(* Logix 5000 project; controller SOCK vendor 1 type 14 code 92 rev 20.56; software revision 20.00 *)

TASK MainTask (periodic, rate 20 ms, priority 10, watchdog 500 ms) : Process

MODULES
   Local : vendor 1 type 14 code 92 (ICP 0, rev 20.56)
      A1_AD2 : vendor 1 type 12 code 200 (ICP 1, Ethernet 172.16.3.121, rev 10.7, Input RPI 500 ms)
      A1_AD3 : vendor 1 type 12 code 200 (Ethernet 172.16.3.123, ICP 2, rev 10.7, Input RPI 500 ms)
END_MODULES

TYPE AcceptResponse :
STRUCT
   Instance : DINT;
   Addr : SockAddr;
END_STRUCT
END_TYPE

TYPE Anpars :
STRUCT
   Tg_inN1 : TAnpar;
   Tg_inAVO1 : TAnpar;
   Tg_outAVO1 : TAnpar;
   Tg_outN1 : TAnpar;
   Tg_inN2 : TAnpar;
   Tg_inAVO2 : TAnpar;
   Tg_outAVO2 : TAnpar;
   Tg_outN2 : TAnpar;
   Pg_aftKr4 : TAnpar;
   Pg_outSep21 : TAnpar;
   Pg_aftKr6 : TAnpar;
   Pg_aftKr16 : TAnpar;
   Pg_outSep22 : TAnpar;
   Pg_aftKr18 : TAnpar;
   dPg_Kr1 : TAnpar;
   dPg_Sep11 : TAnpar;
   dPg_Kr3 : TAnpar;
   dPg_AVO1 : TAnpar;
   dPg_Sep21 : TAnpar;
   dPg_Kr13 : TAnpar;
END_STRUCT
END_TYPE

TYPE OpenConnParam :
STRUCT
   Timeout : DINT;
   DestAddr : STRING;
END_STRUCT
END_TYPE

TYPE READ_DATA_REQ :
STRUCT
   Timeout : DINT;
   BufLen : DINT;
END_STRUCT
END_TYPE

TYPE READ_RESP :
STRUCT
   FromAddr : SockAddr;
   READ_BUFF : STR_4096;
END_STRUCT
END_TYPE

TYPE REQUEST_PARAMETERS :
STRUCT
   Type : DINT;   // 1 - TCP 2- UPD
   Addr : SockAddr;
END_STRUCT
END_TYPE

TYPE SockAddr :
STRUCT
   Family : INT;   // Address Family Must be 2
   Port : INT;   // Port Number
   Addr : DINT;   // IP Address
END_STRUCT
END_TYPE

TYPE SocketData :
STRUCT
   Instance : DINT;
   Attr : SocketInstAttr;
END_STRUCT
END_TYPE

TYPE SocketInstAttr :
STRUCT
   LocalAddr : SockAddr;
   RemoteAddr : SockAddr;
   SendBufSize : DINT;
   RcvBufSize : DINT;
   TCPKeepAlive : DINT;
   TCPNoDelay : DINT;
   InactivityTimeout : DINT;
   MulticastTTL : DINT;
   UDPBroadcast : DINT;
   LingerOnOff : DINT;
END_STRUCT
END_TYPE

TYPE STR_4096 :
STRUCT
   LEN : DINT;
   DATA : SINT[4096];
END_STRUCT
END_TYPE

TYPE STR_480 :
STRUCT
   LEN : DINT;
   DATA : SINT[480];
END_STRUCT
END_TYPE

TYPE TAnpar :
STRUCT
   Sys : REAL;
   Params : INT;
END_STRUCT
END_TYPE

TYPE TFastRetroBuf :
STRUCT
   LEN : DINT;
   PacketSize : DINT;
   Data : REAL[109];
END_STRUCT
END_TYPE

TYPE Write_Data :
STRUCT
   Timeout : DINT;
   ToAddr : SockAddr;
   BufLen : DINT;
   Buf : SINT[20];
END_STRUCT
END_TYPE

TYPE WRT_DATA :
STRUCT
   Timeout : DINT;
   ToAddr : SockAddr;
   Buffer : TFastRetroBuf;
END_STRUCT
END_TYPE

ADD_ON_INSTRUCTION _FastRetro_checkErr   (* revision 1.0 *)
// Проверка ошибок в сообщении, возвращает true, если необходимо предпринять действия
VAR_IN_OUT
   Msg : MESSAGE; {required}
END_VAR
VAR_OUTPUT
   err : DINT; {required}   // Принятие решений 0-не треб., 1-отвалился сокет, 10-другое
END_VAR
VAR_IN_OUT
   errCount : DINT; {required}
END_VAR

ROUTINE Logic   (* structured text *)
   err := 0;
   if(Msg.ER) then
   	if(errCount > 3) then
   		//что-то делаем при ошибке отправки
   		//16#0000_0036 - Соединение принудительно закрыто клиентом, рекоммендация - удалить сокет и поробовать восстановить
   		if(Msg.EXERR = 16#0000_0036
   			or Msg.EXERR = 16#0000_0033 ) then //Обрыв связи
   			err := 1;
   		else
   			err := 10;
   		end_if;
   		//обнуляем хендл соответствующего сокета, так как теперь мы его удаляем (state = 13)
   	end_if;
   else
   	errCount := 0;
   end_if;
END_ROUTINE
END_ADD_ON_INSTRUCTION

ADD_ON_INSTRUCTION _test   (* revision 1.0 *)
// Проверка ошибок в сообщении, возвращает true, если необходимо предпринять действия
VAR_IN_OUT
   Msg : MESSAGE; {required}
END_VAR
VAR_OUTPUT
   err : DINT; {required}   // Принятие решений 0-не треб., 1-отвалился сокет, 10-другое
END_VAR
VAR_IN_OUT
   errCount : DINT; {required}
END_VAR

ROUTINE Logic   (* structured text *)
   err := 0;
   if(Msg.ER) then
   	if(errCount > 3) then
   		//что-то делаем при ошибке отправки
   		//16#0000_0036 - Соединение принудительно закрыто клиентом, рекоммендация - удалить сокет и поробовать восстановить
   		if(Msg.EXERR = 16#0000_0036
   			or Msg.EXERR = 16#0000_0033 ) then //Обрыв связи
   			err := 1;
   		else
   			err := 10;
   		end_if;
   		//обнуляем хендл соответствующего сокета, так как теперь мы его удаляем (state = 13)
   	end_if;
   else
   	errCount := 0;
   end_if;
END_ROUTINE
END_ADD_ON_INSTRUCTION

VAR_GLOBAL   (* controller tags *)
   _EWEB_PATH : STRING := '$01$01';
   AcceptReqTimer : FBD_TIMER;
   Anpar : Anpars;
   BufLenSent : DINT := 7;
   Change_Log_Msg : MESSAGE;
        MessageParameters(ServiceCode := 16#0010, LocalElement := Log_enable, ...)
   CLOCK : DINT[7] := ([0] := 1998, [1] := 1, [2] := 12, [3] := 22, [4] := 11, [5] := 13, [6] := 576094);
   COLN : STRING := ':';
   Conn_Accept_MSG : MESSAGE;
        MessageParameters(ServiceCode := 16#0050, LocalElement := Sock_Accept_Timeout, DestinationTag := Sock_Accept_Resp, ...)
   Create_Sock_MSG : MESSAGE;
        MessageParameters(ServiceCode := 16#004b, LocalElement := Socket, DestinationTag := Instance, ...)
   Delete_All_MSG : MESSAGE;
        MessageParameters(ServiceCode := 16#0051, ...)
   Delete_Sock_MSG : MESSAGE;
        MessageParameters(ServiceCode := 16#004f, ...)
   Enable_Log_MSG : MESSAGE;
        MessageParameters(ServiceCode := 16#000e, DestinationTag := Log_enable, ...)
   Get_Sock_Object_MSG : MESSAGE;
        MessageParameters(ServiceCode := 16#0001, DestinationTag := Socket_Object_Class_Response[0], ...)
   Get_SockTimeout_MSG : MESSAGE;
        MessageParameters(ServiceCode := 16#000e, DestinationTag := SockTimeout, ...)
   HOUR : STRING := '22';
   Instance : DINT := 484;
   Log_enable : DINT;
   Log_old : DINT;
   MINUTE : STRING := '11';
   Read_Data_MSG : MESSAGE;
        MessageParameters(ServiceCode := 16#004d, LocalElement := Read_Data_Req, DestinationTag := Read_Response, ...)
   Read_Data_Req : READ_DATA_REQ := (Timeout := 1000, BufLen := 100);
   Read_Response : READ_RESP := (READ_BUFF := '07:50:1207:50:1307:50:14');
   SECOND : STRING := '13';
   Set_SockTimeout_MSG : MESSAGE;
        MessageParameters(ServiceCode := 16#0010, LocalElement := SockTimeout, ...)
   Sock_Accept_Resp : AcceptResponse := (Instance := 4805, Addr.Family := 2, Addr.Port := 1188, Addr.Addr := 1684298241);
   Sock_Accept_Timeout : DINT := 26000;
   Sock_Object_Data : DINT[13] := ([0] := 655425538, [4] := 2048, [5] := 2048, [6] := 8, [7] := 1, [8] := 300000);
   Socket : REQUEST_PARAMETERS := (Type := 1, Addr.Family := 2, Addr.Port := 10000);
   Socket_Object_Class_Response : SINT[10] := ([0] := 1, [2] := 20);
   SockTimeout : DINT;
   TIME : STRING := '22:11:13';
   Write_Data_MSG : MESSAGE;
        MessageParameters(ServiceCode := 16#004e, LocalElement := Write_Data_Out, DestinationTag := BufLenSent, ...)
   Write_Data_MSG_RED : MESSAGE;
        MessageParameters(ServiceCode := 16#004e, LocalElement := Write_Data_Out, DestinationTag := BufLenSent, ...)
   Write_Data_Out : WRT_DATA := (Timeout := 20000, ToAddr.Family := 2);
   zero : STRING := '0';
END_VAR

PROGRAM _Remove
VAR
   _FastRetro_checkErr : _test;
   Accept : ALIAS FOR Log_Enable.2;
   Accept_Request : BOOL;   // Toggle this Bit to Accept Incoming Connection
   Attrubute : ALIAS FOR Log_Enable.6;
   ClientsId : SocketData[10];
   ClientsIdSize : DINT;
   CommonErrors : DINT;
   ConnCount : DINT;
   Create : ALIAS FOR Log_Enable.0;
   Create_Socket_Req : BOOL;
   CreatedPacketsCount : DINT;
   CurStatusFlagsWrite : DINT;
   CycleNumber : DINT;
   Delete : ALIAS FOR Log_Enable.5;
   Delete_All_Request : BOOL;
   Delete_Sockets_Req : BOOL;
   ElementsCount : DINT;
   Enable_Log_Req : BOOL;
   Err_Write_Red : DINT;
   errCntWriteMain : DINT;
   errCntWriteRed : DINT;
   errCode : DINT;   // Код ошибки
   Errors : ALIAS FOR Log_Enable.7;
   FirstPacketSendMain : BOOL;
   FirstPacketSendRed : BOOL;
   frontSend : BOOL;
   Get_Socket_Instance_Req : BOOL;
   Get_Socket_Object_Req : BOOL;
   Get_SocketTimeout : BOOL;
   increment : DINT;
   isCurSockMain : BOOL;
   it : DINT;
   iter : DINT;
   Log_Enable : DINT := 255;
   loseCyclesCount : DINT;
   MainMsg : DINT; {constant, access Read Only}   // Константа = 0
   MaxCyclesCount : DINT;
   needToResend : BOOL;
   Nothing : BOOL := 1;
   Open : ALIAS FOR Log_Enable.1;
   ParCount : DINT;
   point : REAL;
   Read : ALIAS FOR Log_Enable.3;
   Read_Data_Request : BOOL;   // Toggle This Bit to Read Incoming Data
   RedMsg : DINT := 1; {constant, access Read Only}   // Константа = 1
   SendPacketsCount : DINT;
   serverState : DINT;
   Set_SocketTimeout : BOOL;
   SockInstance : DINT;
   systemDataCount : DINT;
   tcpserverInit : BOOL;
   TempBuffer : REAL[400];
   Write : ALIAS FOR Log_Enable.4;
   Write_Request : BOOL;
END_VAR
END_PROGRAM

PROGRAM MainProgram   (* main routine TCP_Server *)
VAR
   _FastRetro_checkErr : _FastRetro_checkErr;
   Accept : ALIAS FOR Log_Enable.2;
   Accept_Request : BOOL;   // Toggle this Bit to Accept Incoming Connection
   Attrubute : ALIAS FOR Log_Enable.6;
   ClientsId : SocketData[10];
   ClientsIdSize : DINT;
   CommonErrors : DINT;
   ConnCount : DINT;
   Create : ALIAS FOR Log_Enable.0;
   Create_Socket_Req : BOOL;
   CreatedPacketsCount : DINT;
   CurStatusFlagsWrite : DINT;
   CycleNumber : DINT;
   Delete : ALIAS FOR Log_Enable.5;
   Delete_All_Request : BOOL;
   Delete_Sockets_Req : BOOL;
   ElementsCount : DINT;
   Enable_Log_Req : BOOL;
   Err_Write_Red : DINT;
   errCntWriteMain : DINT;
   errCntWriteRed : DINT;
   errCode : DINT;   // Код ошибки
   Errors : ALIAS FOR Log_Enable.7;
   FirstPacketSendMain : BOOL;
   FirstPacketSendRed : BOOL;
   frontSend : BOOL;
   Get_Socket_Instance_Req : BOOL;
   Get_Socket_Object_Req : BOOL;
   Get_SocketTimeout : BOOL;
   increment : DINT;
   isCurSockMain : BOOL;
   it : DINT;
   iter : DINT;
   Log_Enable : DINT := 255;
   loseCyclesCount : DINT;
   MainMsg : DINT; {constant, access Read Only}   // Константа = 0
   MaxCyclesCount : DINT;
   needToResend : BOOL;
   Nothing : BOOL := 1;
   Open : ALIAS FOR Log_Enable.1;
   ParCount : DINT;
   point : REAL;
   Read : ALIAS FOR Log_Enable.3;
   Read_Data_Request : BOOL;   // Toggle This Bit to Read Incoming Data
   RedMsg : DINT := 1; {constant, access Read Only}   // Константа = 1
   SendPacketsCount : DINT;
   serverState : DINT;
   Set_SocketTimeout : BOOL;
   SockInstance : DINT;
   systemDataCount : DINT;
   tcpserverInit : BOOL;
   TempBuffer : REAL[400];
   Write : ALIAS FOR Log_Enable.4;
   Write_Request : BOOL;
END_VAR

ROUTINE _SOCKET_ATTR   (* ladder *)
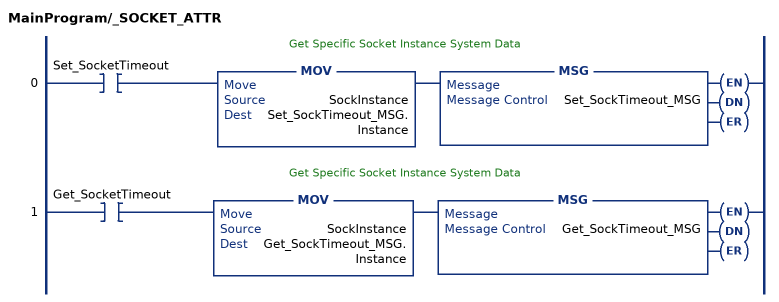
   // Get Specific Socket Instance System Data
   0: XIC(Set_SocketTimeout)MOV(SockInstance,Set_SockTimeout_MSG.Instance)MSG(Set_SockTimeout_MSG);
   // Get Specific Socket Instance System Data
   1: XIC(Get_SocketTimeout)MOV(SockInstance,Get_SockTimeout_MSG.Instance)MSG(Get_SockTimeout_MSG);
END_ROUTINE

ROUTINE _SOCKET_STATS   (* ladder *)
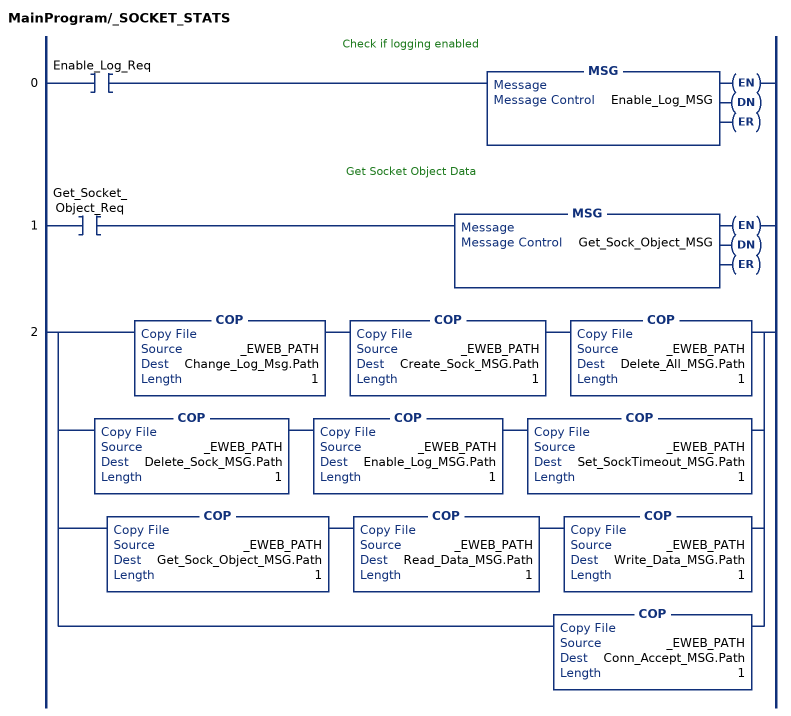
   // Check if logging enabled
   0: XIC(Enable_Log_Req)MSG(Enable_Log_MSG);
   // Get Socket Object Data
   1: XIC(Get_Socket_Object_Req)MSG(Get_Sock_Object_MSG);
   2: [COP(_EWEB_PATH,Change_Log_Msg.Path,1) COP(_EWEB_PATH,Create_Sock_MSG.Path,1) COP(_EWEB_PATH,Delete_All_MSG.Path,1) ,COP(_EWEB_PATH,Delete_Sock_MSG.Path,1) COP(_EWEB_PATH,Enable_Log_MSG.Path,1) COP(_EWEB_PATH,Set_SockTimeout_MSG.Path,1) ,COP(_EWEB_PATH,Get_Sock_Object_MSG.Path,1) COP(_EWEB_PATH,Read_Data_MSG.Path,1) COP(_EWEB_PATH,Write_Data_MSG.Path,1) ,COP(_EWEB_PATH,Conn_Accept_MSG.Path,1) ];
END_ROUTINE

ROUTINE _SOCKET_TCP_SERV   (* ladder *)
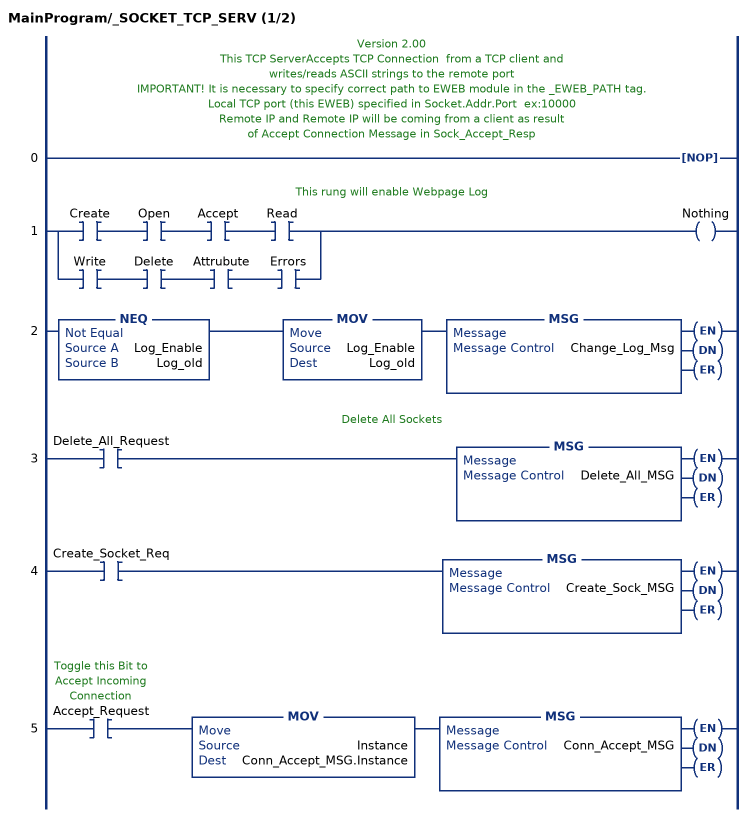
   // Version 2.00
   // This TCP ServerAccepts TCP Connection  from a TCP client and
   // writes/reads ASCII strings to the remote port
   // IMPORTANT! It is necessary to specify correct path to EWEB module in the _EWEB_PATH tag.
   // Local TCP port (this EWEB) specified in Socket.Addr.Port  ex:10000
   // Remote IP and Remote IP will be coming from a client as result
   // of Accept Connection Message in Sock_Accept_Resp
   0: NOP();
   // This rung will enable Webpage Log
   1: [XIC(Create) XIC(Open) XIC(Accept) XIC(Read) ,XIC(Write) XIC(Delete) XIC(Attrubute) XIC(Errors) ]OTE(Nothing);
   2: NEQ(Log_Enable,Log_old)MOV(Log_Enable,Log_old)MSG(Change_Log_Msg);
   // Delete All Sockets
   3: XIC(Delete_All_Request)MSG(Delete_All_MSG);
   4: XIC(Create_Socket_Req)MSG(Create_Sock_MSG);
   5: XIC(Accept_Request)MOV(Instance,Conn_Accept_MSG.Instance)MSG(Conn_Accept_MSG);
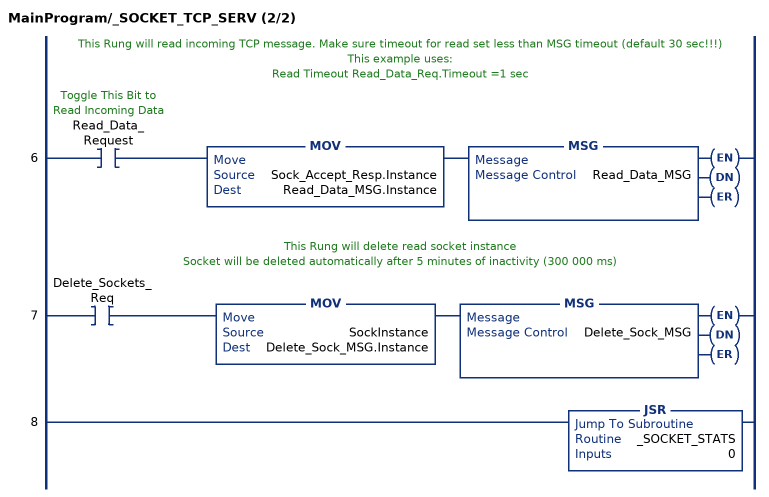
   // This Rung will read incoming TCP message. Make sure timeout for read set less than MSG timeout (default 30 sec!!!)
   // This example uses:
   // Read Timeout Read_Data_Req.Timeout =1 sec
   6: XIC(Read_Data_Request)MOV(Sock_Accept_Resp.Instance,Read_Data_MSG.Instance)MSG(Read_Data_MSG);
   // This Rung will delete read socket instance
   // Socket will be deleted automatically after 5 minutes of inactivity (300 000 ms)
   7: XIC(Delete_Sockets_Req)MOV(SockInstance,Delete_Sock_MSG.Instance)MSG(Delete_Sock_MSG);
   8: JSR(_SOCKET_STATS,0);
END_ROUTINE

ROUTINE _SOCKET_WRITE_MAIN   (* ladder *)
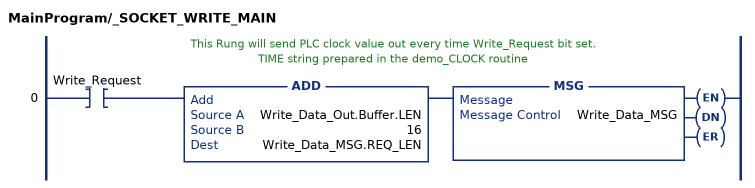
   // This Rung will send PLC clock value out every time Write_Request bit set.
   // TIME string prepared in the demo_CLOCK routine
   0: XIC(Write_Request)ADD(Write_Data_Out.Buffer.LEN,16,Write_Data_MSG.REQ_LEN)MSG(Write_Data_MSG);
END_ROUTINE

ROUTINE _SOCKET_WRITE_RED   (* ladder *)
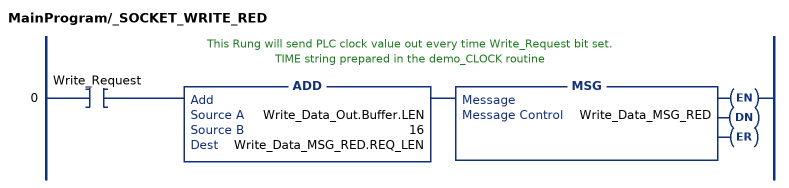
   // This Rung will send PLC clock value out every time Write_Request bit set.
   // TIME string prepared in the demo_CLOCK routine
   0: XIC(Write_Request)ADD(Write_Data_Out.Buffer.LEN,16,Write_Data_MSG_RED.REQ_LEN)MSG(Write_Data_MSG_RED);
END_ROUTINE

ROUTINE Exchange   (* structured text *)
   //Обрабатывается, когда сервер находится в состояниях 2-3
   
   /*
   	Заполнение данных в буфер передачи
   */
   GSV(WALLCLOCKTIME,,DateTime,CLOCK[0]);
   
   //на первом цикле заполняем служебный заголовок пакета
   if(CycleNumber=0) then
   	//дата - год месяц число
   	TempBuffer[0]:= CLOCK[0];
   	TempBuffer[1]:= CLOCK[1];
   	TempBuffer[2]:= CLOCK[2];
   	//время - часы минуты секунды микросекунды
   	TempBuffer[3]:= CLOCK[3];
   	TempBuffer[4]:= CLOCK[4];
   	TempBuffer[5]:= CLOCK[5];
   	TempBuffer[6]:= CLOCK[6];
   	//кол-во параметров
   	TempBuffer[7]:= ParCount;
   	//кол-во циклов для сбора данных
   	TempBuffer[8]:= MaxCyclesCount;
   	(*
   	//дата - год месяц число
   	Write_Data_Out.Buffer.Data[0]:= CLOCK[0];
   	Write_Data_Out.Buffer.Data[1]:= CLOCK[1];
   	Write_Data_Out.Buffer.Data[2]:= CLOCK[2];
   	//время - часы минуты секунды микросекунды
   	Write_Data_Out.Buffer.Data[3]:= CLOCK[3];
   	Write_Data_Out.Buffer.Data[4]:= CLOCK[4];
   	Write_Data_Out.Buffer.Data[5]:= CLOCK[5];
   	Write_Data_Out.Buffer.Data[6]:= CLOCK[6];
   	Write_Data_Out.Buffer.Data[7]:= ParCount;
   	Write_Data_Out.Buffer.Data[8]:= MaxCyclesCount;
   	*)
   end_if;
   
   /*
   ! 	Заполняется пользователем ( правая часть, после := )
   	Порядок следования параметров должен совпадать с описанными в signals.ini (идет в комплекте с FastRetroApp)
   */
   if(CycleNumber<5 and ParCount<=20) then
   	TempBuffer[ParCount*CycleNumber+1+systemDataCount] := Anpar.Tg_inN1.Sys;
   	TempBuffer[ParCount*CycleNumber+2+systemDataCount] := Anpar.Tg_inAVO1.Sys;
   	TempBuffer[ParCount*CycleNumber+3+systemDataCount] := Anpar.Tg_outAVO1.Sys;
   	TempBuffer[ParCount*CycleNumber+4+systemDataCount] := Anpar.Tg_outN1.Sys;
   	TempBuffer[ParCount*CycleNumber+5+systemDataCount] := Anpar.Tg_inN2.Sys;
   	TempBuffer[ParCount*CycleNumber+6+systemDataCount] := Anpar.Tg_inAVO2.Sys;
   	TempBuffer[ParCount*CycleNumber+7+systemDataCount] := Anpar.Tg_outAVO2.Sys;
   	TempBuffer[ParCount*CycleNumber+8+systemDataCount] := Anpar.Tg_outN2.Sys;
   	TempBuffer[ParCount*CycleNumber+9+systemDataCount] := Anpar.Pg_aftKr4.Sys;
   	TempBuffer[ParCount*CycleNumber+10+systemDataCount] := Anpar.Pg_outSep21.Sys;
   	TempBuffer[ParCount*CycleNumber+11+systemDataCount] := Anpar.Pg_aftKr6.Sys;
   	TempBuffer[ParCount*CycleNumber+12+systemDataCount] := Anpar.Pg_aftKr16.Sys;
   	/*
   	TempBuffer[ParCount*CycleNumber+13+systemDataCount] := Anpar.Pg_outSep22.Sys;
   	TempBuffer[ParCount*CycleNumber+14+systemDataCount] := Anpar.Pg_aftKr18.Sys;
   	TempBuffer[ParCount*CycleNumber+15+systemDataCount] := Anpar.dPg_Kr1.Sys;
   	TempBuffer[ParCount*CycleNumber+16+systemDataCount] := Anpar.dPg_Sep11.Sys;
   	TempBuffer[ParCount*CycleNumber+17+systemDataCount] := Anpar.dPg_Kr3.Sys;
   	TempBuffer[ParCount*CycleNumber+18+systemDataCount] := Anpar.dPg_AVO1.Sys;
   	TempBuffer[ParCount*CycleNumber+19+systemDataCount] := Anpar.dPg_Sep21.Sys;
   	TempBuffer[ParCount*CycleNumber+20+systemDataCount] := Anpar.dPg_Kr13.Sys;
   	*/
   else
   	//исп. для отладки
   	loseCyclesCount := loseCyclesCount + 1;
   end_if;
   
   //чтобы предотвратить бесконечный рост CycleNumber
   if(CycleNumber < (MaxCyclesCount + 5)) then
   	CycleNumber := CycleNumber + 1;
   end_if;
   
END_ROUTINE

ROUTINE SendMessage   (* structured text *)
   COP(TempBuffer[0],Write_Data_Out.Buffer.Data[0],ElementsCount);
   //количество сформированных пакетов
   //CreatedPacketsCount := CreatedPacketsCount + 1;
   if(Write_Data_MSG.ER and (ClientsId[MainMsg].Instance>0)) then
   	errCntWriteMain := errCntWriteMain + 1;
   elsif(Write_Data_MSG_RED.ER and (ClientsId[RedMsg].Instance>0)) then
   	errCntWriteRed := errCntWriteRed + 1;
   end_if;
   if(ClientsId[MainMsg].Instance>0) then
   	FirstPacketSendMain := 1;
   end_if;
   if(ClientsId[RedMsg].Instance>0) then
   	FirstPacketSendRed := 1;
   end_if;
   
   Write_Request := 1;
   CycleNumber := 0;
   //NeedToSend.TimerEnable := 0;
   needToResend := 0;
END_ROUTINE

ROUTINE SocketInit   (* structured text *)
   if(isCurSockMain) then
   	SockInstance := ClientsId[MainMsg].Instance;
   else
   	SockInstance := ClientsId[RedMsg].Instance;
   end_if;
   
   //по умолчанию ставим 30 секунд таймаут безактивности
   SockTimeout := 30000;
   Set_SocketTimeout := 1;
   
   JSR(_SOCKET_ATTR);
   
   Set_SocketTimeout := 0;
   
   Get_SocketTimeout := 1;
   JSR(_SOCKET_ATTR);
   Get_SocketTimeout := 0;
END_ROUTINE

ROUTINE TCP_Server   (* structured text *)
   // 	версия 1.0
   /*
   	отправка сообщений асинхронная, поэтому флаги актуально
   	копировать в переменную в начале цикла:
   	.2 - .EW
   	.4 - .ER
   	.5 - .DN
   	.6 - .ST
   	.7 - .EN
   	.8 - .TO
   	.9 - .EN_CC
   */
   CurStatusFlagsWrite := Write_Data_MSG.Flags;
   
   //инициализационные параметры.
   if (not tcpserverInit) then
   
   //! заполняются пользователем
   
   	//количество параметров
   	ParCount := 12;
   //!
   	/*
   		Кол-во циклов в посылке для текущего шага дискретизации.
   		Рекоммендуется отправлять посылки не чаще 100мс, то есть для 20мс цикла вызова задачи значение MaxCyclesCount = 5
   	*/
   	MaxCyclesCount := 5;
   	//размер служебных данных пакета, см. Exchange
   	systemDataCount := 8;
   	//включаем лог
   	Enable_Log_Req := 1;
   	//таймер пересброса ожидания подключения
   	AcceptReqTimer.PRE := 1000;
   
   	SIZE(Write_Data_Out.Buffer.Data,0,ElementsCount);
   
   	//размер посылки данных = (кол-во элементов+служ.параметр) * размер REAL
   	Write_Data_Out.Buffer.LEN := 4*(ElementsCount + 1);
   	Write_Data_Out.Buffer.PacketSize := Write_Data_Out.Buffer.LEN;
   
   	//по клиентам
   	SIZE(ClientsId,0,ClientsIdSize);
   
   	//начальное состояние сервера - создание сокета
   	serverState := 0;
   	tcpserverInit := 1;
   end_if;
   
   TONR(AcceptReqTimer);
   
   /*
   	serverState :=  0 - Инициализация сокета (переход при успехе в 1, иначе в 10)
   					1 - Сокет создан, открываем на прослушку (переход при успехе в 2, иначе в 0)
   					2 - Соединение установлено (одно подключение)
   					3 - Соединение установлено (два подключения)
   					4
   					5
   					10 - Сокет не в норме, очищаем запросы и рестарт (переход при успехе в 0, иначе в 11)
   					11 - Удаляем основной сокет (переход при успехе в 10, иначе в 0)
   					12 - Удаляем сокет прослушки (переход при успехе в 1, иначе повторить)
   					13 - Удаляем сокет прослушки (переход при успехе в 2, иначе повторить)
   
   	ClientsId[MainMsg] - handle сокета MSG
   	ClientsId[RedMsg] - handle сокета MSG_RED
   */
   CASE serverState OF
   
   0:
   	if(not Create_Socket_Req) then
   		Create_Socket_Req := 1;
   	elsif(Create_Sock_MSG.EN) then
   	  if(Create_Sock_MSG.DN) then
   		Create_Socket_Req := 0;
   		ConnCount := 0;
   		serverState := 1;
   	  elsif(Create_Sock_MSG.ER) then
   	  	Create_Socket_Req := 0;
   		if(Create_Sock_MSG.EXERR = 16#0000_0030) then
   			//повторное создание сокета, попробуем пересоздать
   			serverState := 10;
   		end_if;
   	  end_if;
   	end_if;
   
   1:
   	loseCyclesCount := 0;
   	CreatedPacketsCount := 0;
   	SendPacketsCount := 0;
   	errCntWriteMain := 0;
   	errCntWriteRed := 0;
   	CommonErrors := 0;
   	FirstPacketSendRed := 0;
   	FirstPacketSendMain := 0;
   
   	//Взводим секундный таймер, по истечение которого начинаем слушать сокет на новые подключения
   	if(not Accept_Request ) then
   		AcceptReqTimer.TimerEnable := 1;
   		Accept_Request := AcceptReqTimer.DN;
   	elsif( Conn_Accept_MSG.DN) then
   		//при успешном подключении нового клиента переходим в состояние 2
   		FOR iter := 0 TO ClientsIdSize-1 DO
   			ClientsId[iter].Instance := 0;
   		END_FOR;
   		ClientsId[MainMsg].Instance := Sock_Accept_Resp.Instance;
   		Accept_Request := 0;
   		AcceptReqTimer.TimerEnable := 0;
   		serverState := 2;
   		isCurSockMain := 1;
   		//инициализация таймаута инактивности по новому соединению
   		JSR(SocketInit);
   	elsif(Conn_Accept_MSG.ER) then
   		Accept_Request := 0;
   		AcceptReqTimer.TimerEnable := 0;
   		if(Conn_Accept_MSG.ERR = 16#0005) then //сокет был закрыт по неактивности
   			serverState := 0;
   		end_if;
   	end_if;
   2:
   	//обработка подключения резервного клиента
   	if(not Accept_Request ) then
   		AcceptReqTimer.TimerEnable := 1;
   		Accept_Request := AcceptReqTimer.DN;
   	elsif( Conn_Accept_MSG.DN) then
   		/*
   			если подключился второй клиент - запоминаем его Instance в пустую в текущий момент структуру,
   			т.к. мы точно не знаем, какой из клиентов отвалился, если мы были в state = 3 (основной или резервный)
   		*/
   		if(ClientsId[RedMsg].Instance = 0) then
   			ClientsId[RedMsg].Instance := Sock_Accept_Resp.Instance;
   			serverState := 3;
   			//переменная используется в SocketInit
   			isCurSockMain := 0;
   			JSR(SocketInit);
   		elsif(ClientsId[MainMsg].Instance = 0) then
   			ClientsId[MainMsg].Instance := Sock_Accept_Resp.Instance;
   			serverState := 3;
   			isCurSockMain := 1;
   			JSR(SocketInit);
   		end_if;
   		Accept_Request := 0;
   	elsif(Conn_Accept_MSG.ER) then
   		Accept_Request := 0;
   		AcceptReqTimer.TimerEnable := 0;
   		if(Conn_Accept_MSG.ERR = 16#0005) then //сокет был закрыт по неактивности
   			serverState := 0;
   		end_if;
   	end_if;
   
   	if((ClientsId[MainMsg].Instance>0) and (ClientsId[RedMsg].Instance>0)) then
   		serverState := 3;
   	end_if;
   	if(CycleNumber>=MaxCyclesCount or needToResend) then
   		//отправляем пакет...
   		JSR(SendMessage);
   	else
   		Write_Request := 0;
   	end_if;
   	//обработка обмена
   	JSR(Exchange);
   
   	/*
   		Обработка ошибок отправки.
   		1. FirstPacketSendMain (Red) - признак того, что по соответсвующему соединению был отправлен пакет.
   		Необходимо контролировать, так как, флаг MSG - .ER хранится в неактивном состоянии, и сбрасывается лишь при
   		пересбросе флага .EN, то есть контрольного бита управляющей цепочки, в данном случае Write_Request
   		2. needToResend - флаг необходимости повторной отправки сообщения. Не используется, так как возможны зацикливания
   		системы, если ошибка фундаментальная. Лучше пропустить пакет, чем повесить весь обмен.
   		3._FastRetro_checkErr выдает тип ошибки, если она повторилась опр. число раз (см. код _FastRetro_checkErr)
   
   		В общем случае, если код, выданный _FastRetro_checkErr <> 0, то переходим в состояние 12 (пересоздаем текущий локальный сокет)
   	*/
   	if((ClientsId[MainMsg].Instance>0) and FirstPacketSendMain) then
   		_FastRetro_checkErr(_FastRetro_checkErr,Write_Data_MSG,errCode,errCntWriteMain);
   		if(errCode > 0) then
   			point := point + 1;
   			FirstPacketSendMain := 0;
   			SockInstance := Write_Data_MSG.Instance;
   			ClientsId[MainMsg].Instance := 0;
   			serverState := 12;
   		else
   			;//needToResend := 1;
   		end_if;
   
   	elsif((ClientsId[RedMsg].Instance>0) and FirstPacketSendRed) then
   		_FastRetro_checkErr(_FastRetro_checkErr,Write_Data_MSG_RED,errCode,errCntWriteRed);
   		if(errCode > 0) then
   			FirstPacketSendRed := 0;
   			SockInstance := Write_Data_MSG_RED.Instance;
   			ClientsId[RedMsg].Instance := 0;
   			serverState := 12;
   		else
   			;//needToResend := 1;
   		end_if;
   	end_if;
   
   3:	//Работает и основное и резервное соединение
   	if(CycleNumber>=MaxCyclesCount or needToResend) then
   		//отправляем пакет...
   		JSR(SendMessage);
   	else
   		Write_Request := 0;
   	end_if;
   
   	JSR(Exchange);
   
   	if(Write_Data_MSG.ER and FirstPacketSendMain or Write_Data_MSG_RED.ER and FirstPacketSendRed) then
   		//если ошибка при отправке основного сообщения
   		if((errCntWriteMain > 3) and (ClientsId[MainMsg].Instance>0)) then
   			_FastRetro_checkErr(_FastRetro_checkErr,Write_Data_MSG,errCode,errCntWriteMain);
   			if(errCode > 0) then
   				FirstPacketSendMain := 0;
   				SockInstance := Write_Data_MSG.Instance;
   				//обнуляем хендл соответствующего сокета, так как теперь мы его удаляем (state = 13)
   				ClientsId[MainMsg].Instance := 0;
   				serverState := 13;
   			else
   				;//needToResend := 1;
   			end_if;
   		elsif((errCntWriteRed > 3) and (ClientsId[RedMsg].Instance>0)) then
   			_FastRetro_checkErr(_FastRetro_checkErr,Write_Data_MSG_RED,errCode,errCntWriteRed);
   			if(errCode > 0) then
   				FirstPacketSendRed := 0;
   				SockInstance := Write_Data_MSG_RED.Instance;
   				//обнуляем хендл соответствующего сокета, так как теперь мы его удаляем (state = 13)
   				ClientsId[RedMsg].Instance := 0;
   				serverState := 13;
   			else
   				;//needToResend := 1;
   			end_if;
   		end_if;
   			//что-то делаем при ошибке отправки
   			//16#0000_0036 - Соединение принудительно закрыто клиентом, рекоммендация - удалить сокет и поробовать восстановить
   
   	end_if;
   
   10:
   	if(not Delete_All_Request) then
   		Delete_All_Request := 1;
   	elsif(Delete_All_MSG.DN) then
   		Delete_All_Request := 0;
   		serverState := 0;
   	elsif(Delete_All_MSG.ER) then
   		Delete_All_Request := 0;
   		serverState := 11;
   	end_if;
   
   11:
   	SockInstance := Instance;
   	if(not Delete_Sockets_Req) then
   		Delete_Sockets_Req := 1;
   	elsif(Delete_Sock_MSG.DN) then
   		Delete_Sockets_Req := 0;
   		serverState := 10;
   	elsif(Delete_Sock_MSG.ER) then
   		if(Delete_Sock_MSG.ERR = 16#0005) then
   			serverState := 0;
   		else
   			Delete_Sockets_Req := 0;
   		end_if;
   	end_if;
   
   12:
   	//SockInstance := Sock_Accept_Resp.Instance;
   	if(not Delete_Sockets_Req) then
   		Delete_Sockets_Req := 1;
   	elsif(Delete_Sock_MSG.DN or (Delete_Sock_MSG.ERR = 16#0005)) then
   		Delete_Sockets_Req := 0;
   		serverState := 1;
   	elsif(Delete_Sock_MSG.ER) then
   		Delete_Sockets_Req := 0;
   	end_if;
   13:
   	//SockInstance := Sock_Accept_Resp.Instance;
   	if(not Delete_Sockets_Req) then
   		Delete_Sockets_Req := 1;
   	elsif(Delete_Sock_MSG.DN) then
   		Delete_Sockets_Req := 0;
   		serverState := 2;
   	elsif(Delete_Sock_MSG.ER) then
   		Delete_Sockets_Req := 0;
   	end_if;
   
   END_CASE;
   
   
   //обработка сокета
   JSR(_SOCKET_TCP_SERV);
   
   if(ClientsId[MainMsg].Instance>0) then
   	Write_Data_MSG.Instance := ClientsId[MainMsg].Instance;
   	JSR(_SOCKET_WRITE_MAIN);
   end_if;
   if(ClientsId[RedMsg].Instance>0) then
   	Write_Data_MSG_RED.Instance := ClientsId[RedMsg].Instance;
   	JSR(_SOCKET_WRITE_RED);
   end_IF;
   
   
   
   
   
END_ROUTINE
END_PROGRAM

PROGRAM Process   (* main routine imit *)
VAR
   countDistort : DINT;
   Init : BOOL;
   oldVal : REAL;
   reverse : INT;
END_VAR

ROUTINE imit   (* structured text *)
   if (not Init) then
   	reverse := 1;
   	Init := 1;
   	countDistort := 0;
   end_if;
   
   GSV(WALLCLOCKTIME,,DateTime,CLOCK[0]);
   
   reverse := -1*reverse;
   
   oldVal := Anpar.Tg_inN1.Sys;
   Anpar.Tg_inN1.Sys := Anpar.Tg_inN1.Sys + 1;
   if(ABS(Anpar.Tg_inN1.Sys - oldVal) > 2) then countDistort := countDistort + 1; END_IF;
   if(Anpar.Tg_inN1.Sys > 50) then Anpar.Tg_inN1.Sys := -50; END_IF;
   
   Anpar.Tg_inAVO1.Sys := CLOCK[5] + reverse*CLOCK[6]/10000 + 20;
   Anpar.Tg_outAVO1.Sys := CLOCK[5] + reverse*CLOCK[6]/10000 + 30;
   Anpar.Tg_outN1.Sys := CLOCK[5] + reverse*CLOCK[6]/10000 + 40;
   Anpar.Tg_inN2.Sys := CLOCK[5] + reverse*CLOCK[6]/10000 + 50;
   Anpar.Tg_inAVO2.Sys := CLOCK[5] + reverse*CLOCK[6]/10000 + 60;
   Anpar.Tg_outAVO2.Sys := CLOCK[5] + reverse*CLOCK[6]/10000 + 70;
   Anpar.Tg_outN2.Sys := CLOCK[5] + reverse*CLOCK[6]/10000 + 80;
   Anpar.Pg_aftKr4.Sys := CLOCK[5] + reverse*CLOCK[6]/10000 + 90;
   Anpar.Pg_outSep21.Sys := CLOCK[5] + reverse*CLOCK[6]/10000 + 100;
   Anpar.Pg_aftKr6.Sys := CLOCK[5] + reverse*CLOCK[6]/10000 + 110;
   Anpar.Pg_aftKr16.Sys := CLOCK[5] + reverse*CLOCK[6]/10000 + 120;
   Anpar.Pg_outSep22.Sys := CLOCK[5] + reverse*CLOCK[6]/10000 + 130;
   Anpar.Pg_aftKr18.Sys := CLOCK[5] + reverse*CLOCK[6]/10000 + 140;
   Anpar.dPg_Kr1.Sys := CLOCK[5] + reverse*CLOCK[6]/10000 + 150;
   Anpar.dPg_Sep11.Sys := CLOCK[5] + reverse*CLOCK[6]/10000 + 160;
   Anpar.dPg_Kr3.Sys := CLOCK[5] + reverse*CLOCK[6]/10000 + 170;
   Anpar.dPg_AVO1.Sys := CLOCK[5] + reverse*CLOCK[6]/10000 + 180;
   Anpar.dPg_Sep21.Sys := CLOCK[5] + reverse*CLOCK[6]/10000 + 190;
   Anpar.dPg_Kr13.Sys := CLOCK[5] + reverse*CLOCK[6]/10000 + 200;
   
   
END_ROUTINE
END_PROGRAM
